{attribute 'qualified_only'}
VAR_GLOBAL
		EtherCAT_Master_ELxxxx : EtherCAT_Master_ELxxxx_D0BA48C6;
END_VAR

(* stored: Version 1.2.0.0, ProductVersion 3.1.4024.11
   GVL GVL_iXlinker: Id {62ed5de5-995a-48b8-924c-6b6653cee977} *)
